FUNCTION_BLOCK GENERATE_TWO_RANDOM
  {SET_ATTRIBUTE(OpcUa, SERVICE)}
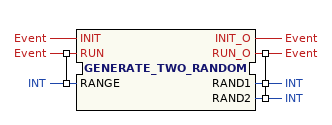
  EVENT_INPUT
    INIT;
    RUN WITH RANGE; {SET_ATTRIBUTE(OpcUa, Method)}
  END_EVENT
  EVENT_OUTPUT
    INIT_O;
    RUN_O WITH RAND1, RAND2;
  END_EVENT
  VAR_INPUT
    RANGE : INT; {SET_ATTRIBUTE(OpcUa, Constant.RUN)}
  END_VAR
  VAR_OUTPUT
    RAND1 : INT; {SET_ATTRIBUTE(OpcUa, Variable.RUN_O)}
    RAND2 : INT; {SET_ATTRIBUTE(OpcUa, Variable.RUN_O)}
  END_VAR
END_FUNCTION_BLOCK
